// Mitsubishi GX Works2 project: DALG_TRAM_BE_TONG_ANALOG   PLC: FX3U/FX3UC

PROGRAM MAIN
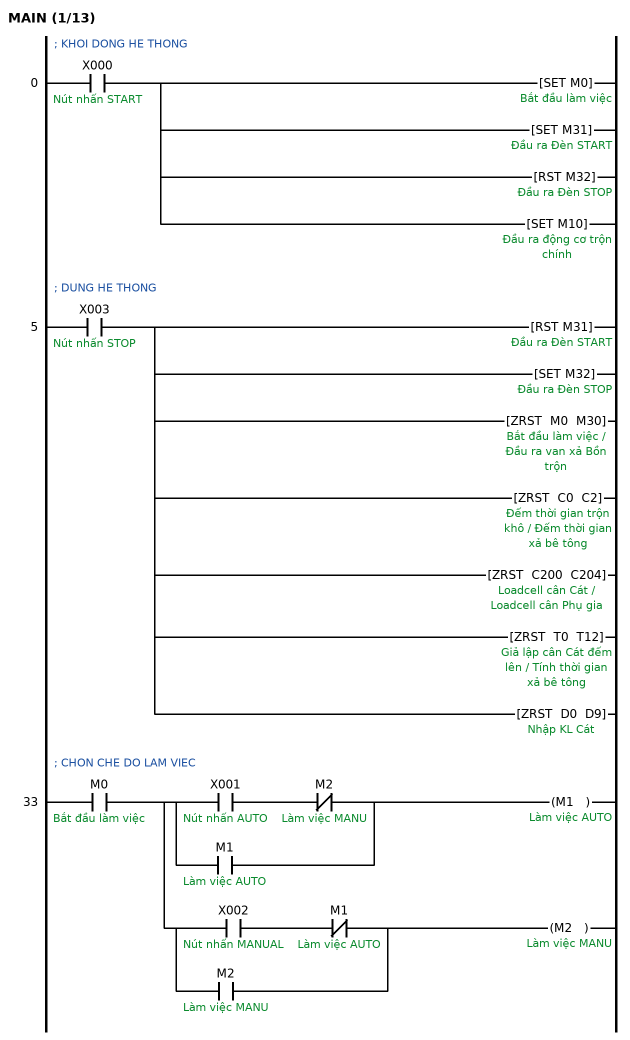
; KHOI DONG HE THONG
0     LD      X000  ; Nút nhấn START
      SET     M0  ; Bắt đầu làm việc
      SET     M31  ; Đầu ra Đèn START
      RST     M32  ; Đầu ra Đèn STOP
      SET     M10  ; Đầu ra động cơ trộn chính
; DUNG HE THONG
5     LD      X003  ; Nút nhấn STOP
      RST     M31  ; Đầu ra Đèn START
      SET     M32  ; Đầu ra Đèn STOP
      ZRST    M0 M30  ; Đầu ra van xả Bồn trộn
      ZRST    C0 C2  ; Đếm thời gian trộn khô / Đếm thời gian xả bê tông
      ZRST    C200 C204  ; Loadcell cân Cát / Loadcell cân Phụ gia
      ZRST    T0 T12  ; Giả lập cân Cát đếm lên / Tính thời gian xả bê tông
      ZRST    D0 D9  ; Nhập KL Cát
; CHON CHE DO LAM VIEC
33    LD      M0  ; Bắt đầu làm việc
      MPS
      LD      X001  ; Nút nhấn AUTO
      ANI     M2  ; Làm việc MANU
      OR      M1  ; Làm việc AUTO
      ANB
      OUT     M1  ; Làm việc AUTO
      MPP
      LD      X002  ; Nút nhấn MANUAL
      ANI     M1  ; Làm việc AUTO
      OR      M2  ; Làm việc MANU
      ANB
      OUT     M2  ; Làm việc MANU
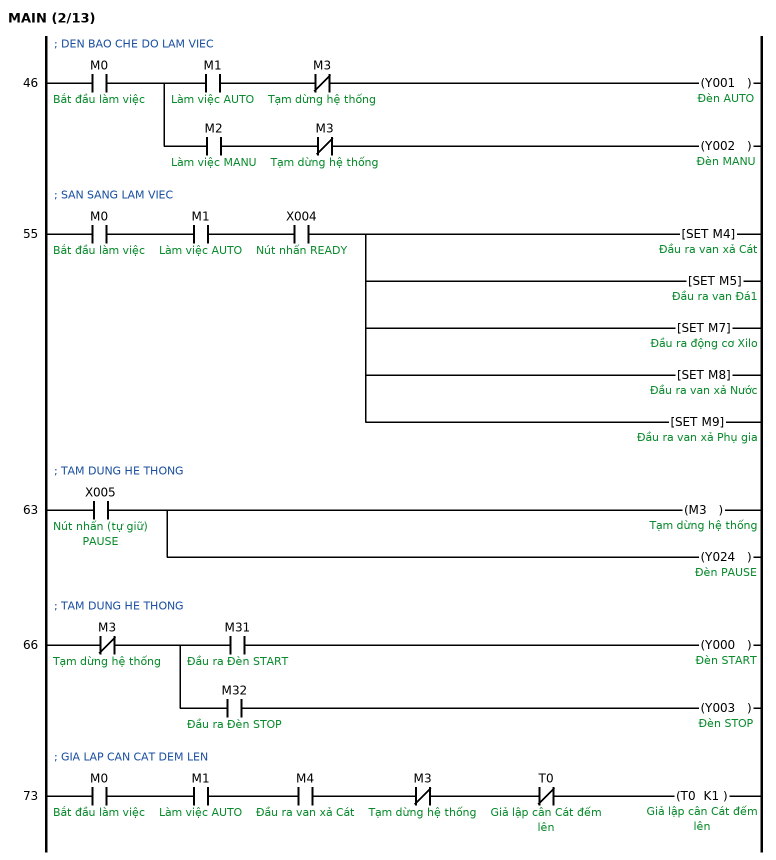
; DEN BAO CHE DO LAM VIEC
46    LD      M0  ; Bắt đầu làm việc
      MPS
      AND     M1  ; Làm việc AUTO
      ANI     M3  ; Tạm dừng hệ thống
      OUT     Y001  ; Đèn AUTO
      MPP
      AND     M2  ; Làm việc MANU
      ANI     M3  ; Tạm dừng hệ thống
      OUT     Y002  ; Đèn MANU
; SAN SANG LAM VIEC
55    LD      M0  ; Bắt đầu làm việc
      AND     M1  ; Làm việc AUTO
      AND     X004  ; Nút nhấn READY
      SET     M4  ; Đầu ra van xả Cát
      SET     M5  ; Đầu ra van Đá1
      SET     M7  ; Đầu ra động cơ Xilo
      SET     M8  ; Đầu ra van xả Nước
      SET     M9  ; Đầu ra van xả Phụ gia
; TAM DUNG HE THONG
63    LD      X005  ; Nút nhấn (tự giữ) PAUSE
      OUT     M3  ; Tạm dừng hệ thống
      OUT     Y024  ; Đèn PAUSE
; TAM DUNG HE THONG
66    LDI     M3  ; Tạm dừng hệ thống
      MPS
      AND     M31  ; Đầu ra Đèn START
      OUT     Y000  ; Đèn START
      MPP
      AND     M32  ; Đầu ra Đèn STOP
      OUT     Y003  ; Đèn STOP
; GIA LAP CAN CAT DEM LEN
73    LD      M0  ; Bắt đầu làm việc
      AND     M1  ; Làm việc AUTO
      AND     M4  ; Đầu ra van xả Cát
      ANI     M3  ; Tạm dừng hệ thống
      ANI     T0  ; Giả lập cân Cát đếm lên
      OUT     T0 K1  ; Giả lập cân Cát đếm lên
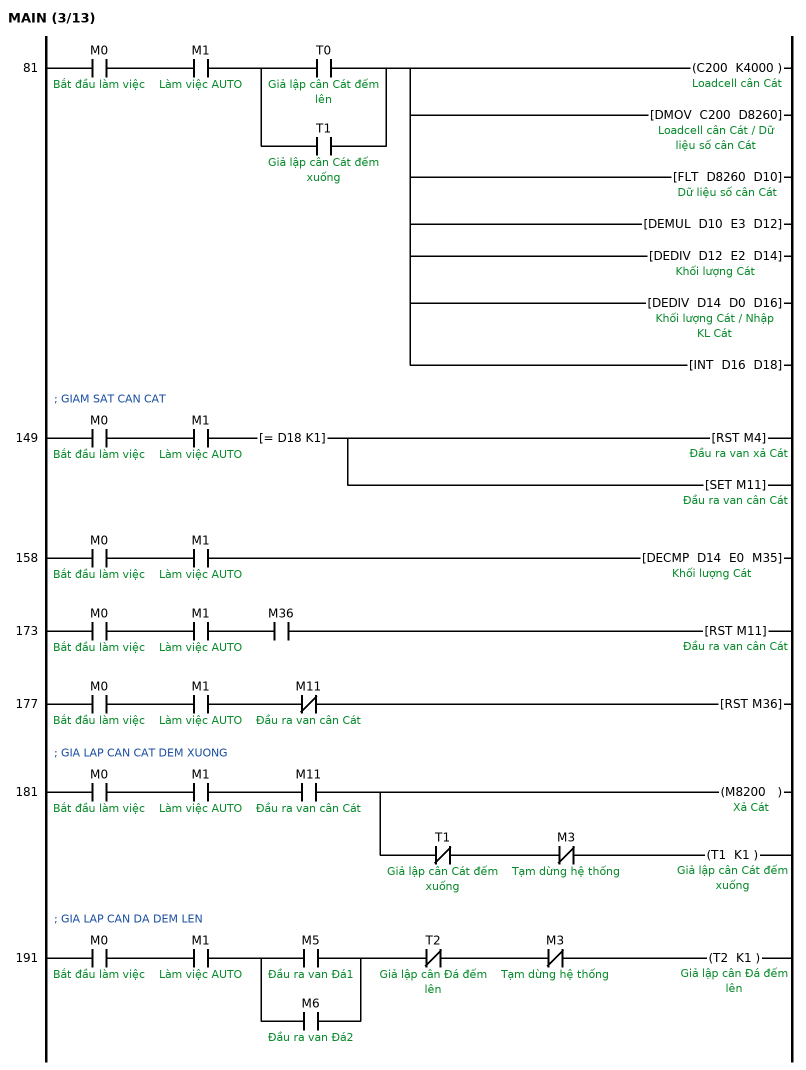
81    LD      M0  ; Bắt đầu làm việc
      AND     M1  ; Làm việc AUTO
      LD      T0  ; Giả lập cân Cát đếm lên
      OR      T1  ; Giả lập cân Cát đếm xuống
      ANB
      OUT     C200 K4000  ; Loadcell cân Cát
      DMOV    C200 D8260  ; Dữ liệu số cân Cát
      FLT     D8260 D10
      DEMUL   D10 E3 D12
      DEDIV   D12 E2 D14  ; Khối lượng Cát
      DEDIV   D14 D0 D16
      INT     D16 D18
; GIAM SAT CAN CAT
149   LD      M0  ; Bắt đầu làm việc
      AND     M1  ; Làm việc AUTO
      AND=    D18 K1
      RST     M4  ; Đầu ra van xả Cát
      SET     M11  ; Đầu ra van cân Cát
158   LD      M0  ; Bắt đầu làm việc
      AND     M1  ; Làm việc AUTO
      DECMP   D14 E0 M35
173   LD      M0  ; Bắt đầu làm việc
      AND     M1  ; Làm việc AUTO
      AND     M36
      RST     M11  ; Đầu ra van cân Cát
177   LD      M0  ; Bắt đầu làm việc
      AND     M1  ; Làm việc AUTO
      ANI     M11  ; Đầu ra van cân Cát
      RST     M36
; GIA LAP CAN CAT DEM XUONG
181   LD      M0  ; Bắt đầu làm việc
      AND     M1  ; Làm việc AUTO
      AND     M11  ; Đầu ra van cân Cát
      OUT     M8200  ; Xả Cát
      ANI     T1  ; Giả lập cân Cát đếm xuống
      ANI     M3  ; Tạm dừng hệ thống
      OUT     T1 K1  ; Giả lập cân Cát đếm xuống
; GIA LAP CAN DA DEM LEN
191   LD      M0  ; Bắt đầu làm việc
      AND     M1  ; Làm việc AUTO
      LD      M5  ; Đầu ra van Đá1
      OR      M6  ; Đầu ra van Đá2
      ANB
      ANI     T2  ; Giả lập cân Đá đếm lên
      ANI     M3  ; Tạm dừng hệ thống
      OUT     T2 K1  ; Giả lập cân Đá đếm lên
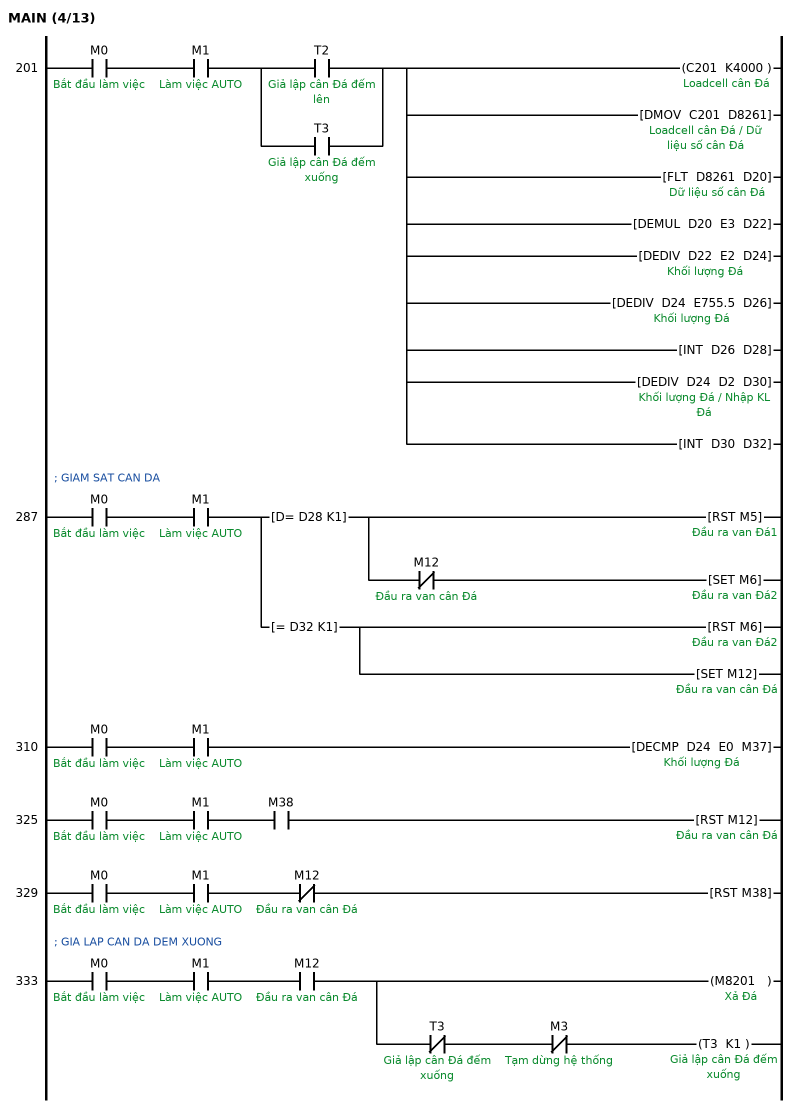
201   LD      M0  ; Bắt đầu làm việc
      AND     M1  ; Làm việc AUTO
      LD      T2  ; Giả lập cân Đá đếm lên
      OR      T3  ; Giả lập cân Đá đếm xuống
      ANB
      OUT     C201 K4000  ; Loadcell cân Đá
      DMOV    C201 D8261  ; Dữ liệu số cân Đá
      FLT     D8261 D20
      DEMUL   D20 E3 D22
      DEDIV   D22 E2 D24  ; Khối lượng Đá
      DEDIV   D24 E755.5 D26
      INT     D26 D28
      DEDIV   D24 D2 D30  ; Nhập KL Đá
      INT     D30 D32
; GIAM SAT CAN DA
287   LD      M0  ; Bắt đầu làm việc
      AND     M1  ; Làm việc AUTO
      MPS
      ANDD=   D28 K1
      RST     M5  ; Đầu ra van Đá1
      ANI     M12  ; Đầu ra van cân Đá
      SET     M6  ; Đầu ra van Đá2
      MPP
      AND=    D32 K1
      RST     M6  ; Đầu ra van Đá2
      SET     M12  ; Đầu ra van cân Đá
310   LD      M0  ; Bắt đầu làm việc
      AND     M1  ; Làm việc AUTO
      DECMP   D24 E0 M37
325   LD      M0  ; Bắt đầu làm việc
      AND     M1  ; Làm việc AUTO
      AND     M38
      RST     M12  ; Đầu ra van cân Đá
329   LD      M0  ; Bắt đầu làm việc
      AND     M1  ; Làm việc AUTO
      ANI     M12  ; Đầu ra van cân Đá
      RST     M38
; GIA LAP CAN DA DEM XUONG
333   LD      M0  ; Bắt đầu làm việc
      AND     M1  ; Làm việc AUTO
      AND     M12  ; Đầu ra van cân Đá
      OUT     M8201  ; Xả Đá
      ANI     T3  ; Giả lập cân Đá đếm xuống
      ANI     M3  ; Tạm dừng hệ thống
      OUT     T3 K1  ; Giả lập cân Đá đếm xuống
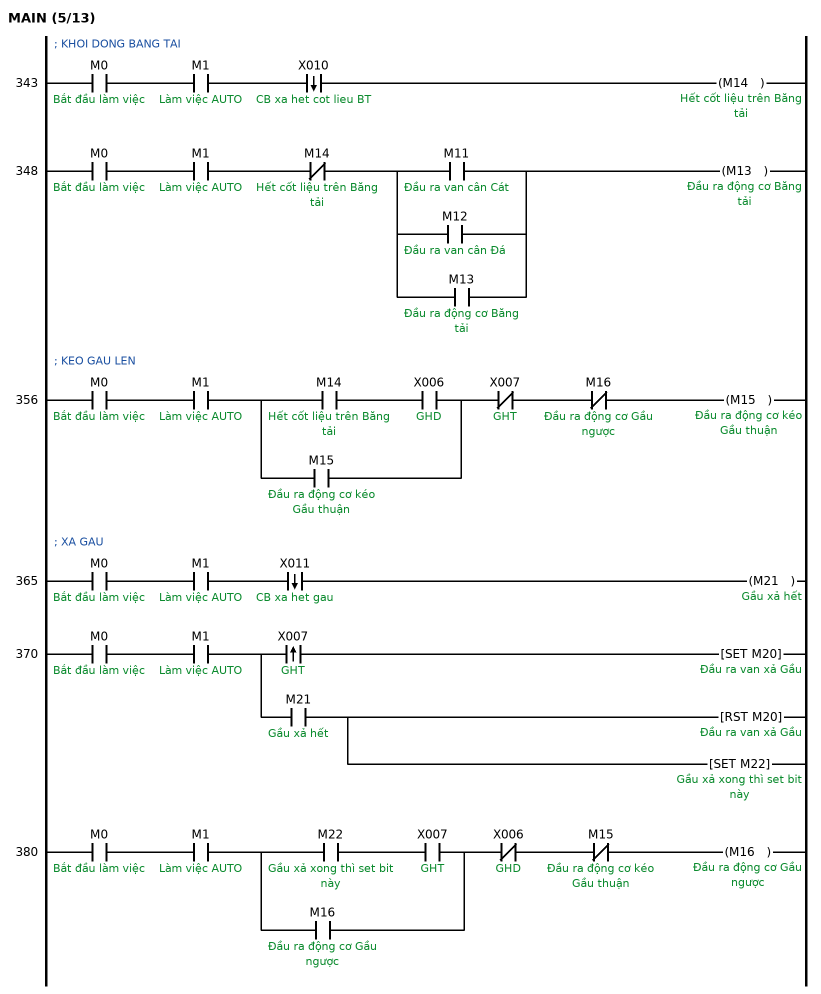
; KHOI DONG BANG TAI
343   LD      M0  ; Bắt đầu làm việc
      AND     M1  ; Làm việc AUTO
      ANDF    X010  ; CB xa het cot lieu BT
      OUT     M14  ; Hết cốt liệu trên Băng tải
348   LD      M0  ; Bắt đầu làm việc
      AND     M1  ; Làm việc AUTO
      ANI     M14  ; Hết cốt liệu trên Băng tải
      LD      M11  ; Đầu ra van cân Cát
      OR      M12  ; Đầu ra van cân Đá
      OR      M13  ; Đầu ra động cơ Băng tải
      ANB
      OUT     M13  ; Đầu ra động cơ Băng tải
; KEO GAU LEN
356   LD      M0  ; Bắt đầu làm việc
      AND     M1  ; Làm việc AUTO
      LD      M14  ; Hết cốt liệu trên Băng tải
      AND     X006  ; GHD
      OR      M15  ; Đầu ra động cơ kéo Gầu thuận
      ANB
      ANI     X007  ; GHT
      ANI     M16  ; Đầu ra động cơ Gầu ngược
      OUT     M15  ; Đầu ra động cơ kéo Gầu thuận
; XA GAU
365   LD      M0  ; Bắt đầu làm việc
      AND     M1  ; Làm việc AUTO
      ANDF    X011  ; CB xa het gau
      OUT     M21  ; Gầu xả hết
370   LD      M0  ; Bắt đầu làm việc
      AND     M1  ; Làm việc AUTO
      MPS
      ANDP    X007  ; GHT
      SET     M20  ; Đầu ra van xả Gầu
      MPP
      AND     M21  ; Gầu xả hết
      RST     M20  ; Đầu ra van xả Gầu
      SET     M22  ; Gầu xả xong thì set bit này
380   LD      M0  ; Bắt đầu làm việc
      AND     M1  ; Làm việc AUTO
      LD      M22  ; Gầu xả xong thì set bit này
      AND     X007  ; GHT
      OR      M16  ; Đầu ra động cơ Gầu ngược
      ANB
      ANI     X006  ; GHD
      ANI     M15  ; Đầu ra động cơ kéo Gầu thuận
      OUT     M16  ; Đầu ra động cơ Gầu ngược
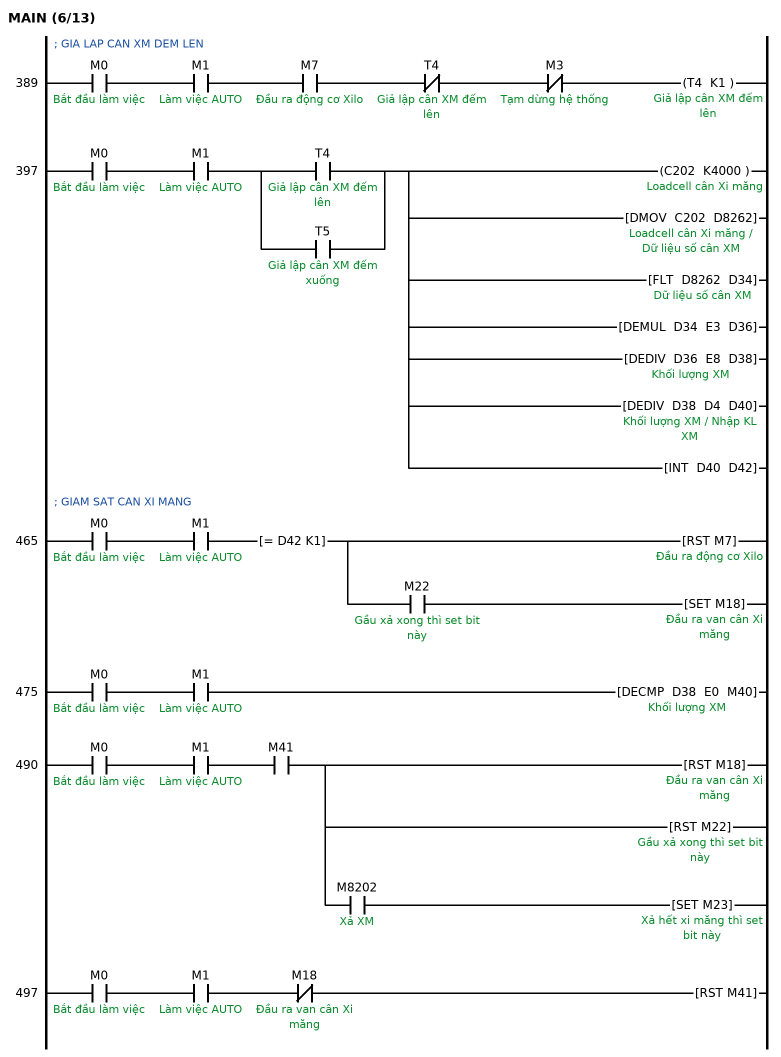
; GIA LAP CAN XM DEM LEN
389   LD      M0  ; Bắt đầu làm việc
      AND     M1  ; Làm việc AUTO
      AND     M7  ; Đầu ra động cơ Xilo
      ANI     T4  ; Giả lập cân XM đếm lên
      ANI     M3  ; Tạm dừng hệ thống
      OUT     T4 K1  ; Giả lập cân XM đếm lên
397   LD      M0  ; Bắt đầu làm việc
      AND     M1  ; Làm việc AUTO
      LD      T4  ; Giả lập cân XM đếm lên
      OR      T5  ; Giả lập cân XM đếm xuống
      ANB
      OUT     C202 K4000  ; Loadcell cân Xi măng
      DMOV    C202 D8262  ; Dữ liệu số cân XM
      FLT     D8262 D34
      DEMUL   D34 E3 D36
      DEDIV   D36 E8 D38  ; Khối lượng XM
      DEDIV   D38 D4 D40  ; Nhập KL XM
      INT     D40 D42
; GIAM SAT CAN XI MANG
465   LD      M0  ; Bắt đầu làm việc
      AND     M1  ; Làm việc AUTO
      AND=    D42 K1
      RST     M7  ; Đầu ra động cơ Xilo
      AND     M22  ; Gầu xả xong thì set bit này
      SET     M18  ; Đầu ra van cân Xi măng
475   LD      M0  ; Bắt đầu làm việc
      AND     M1  ; Làm việc AUTO
      DECMP   D38 E0 M40
490   LD      M0  ; Bắt đầu làm việc
      AND     M1  ; Làm việc AUTO
      AND     M41
      RST     M18  ; Đầu ra van cân Xi măng
      RST     M22  ; Gầu xả xong thì set bit này
      AND     M8202  ; Xả XM
      SET     M23  ; Xả hết xi măng thì set bit này
497   LD      M0  ; Bắt đầu làm việc
      AND     M1  ; Làm việc AUTO
      ANI     M18  ; Đầu ra van cân Xi măng
      RST     M41
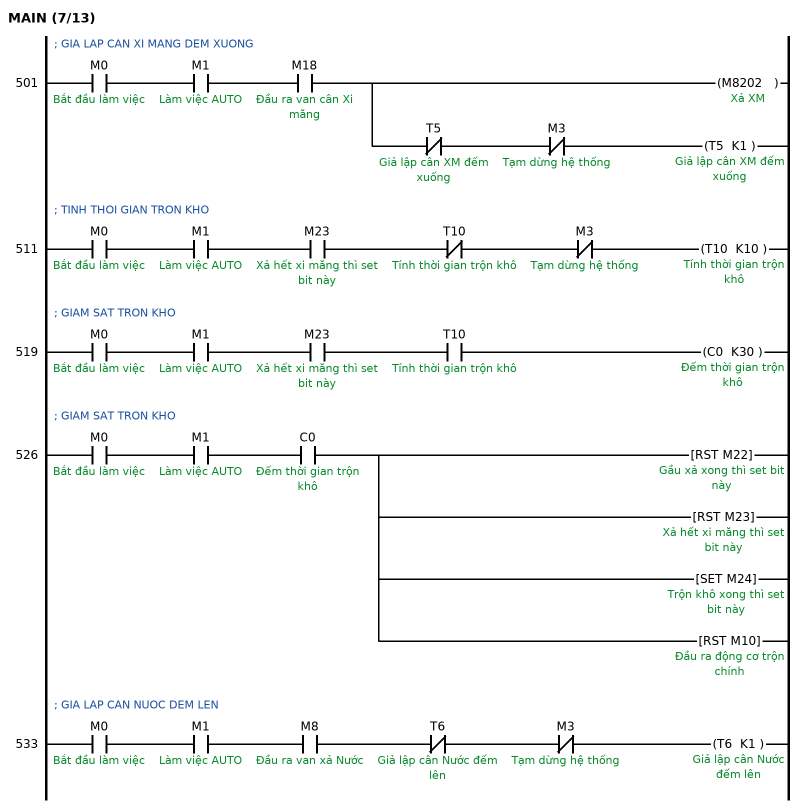
; GIA LAP CAN XI MANG DEM XUONG
501   LD      M0  ; Bắt đầu làm việc
      AND     M1  ; Làm việc AUTO
      AND     M18  ; Đầu ra van cân Xi măng
      OUT     M8202  ; Xả XM
      ANI     T5  ; Giả lập cân XM đếm xuống
      ANI     M3  ; Tạm dừng hệ thống
      OUT     T5 K1  ; Giả lập cân XM đếm xuống
; TINH THOI GIAN TRON KHO
511   LD      M0  ; Bắt đầu làm việc
      AND     M1  ; Làm việc AUTO
      AND     M23  ; Xả hết xi măng thì set bit này
      ANI     T10  ; Tính thời gian trộn khô
      ANI     M3  ; Tạm dừng hệ thống
      OUT     T10 K10  ; Tính thời gian trộn khô
; GIAM SAT TRON KHO
519   LD      M0  ; Bắt đầu làm việc
      AND     M1  ; Làm việc AUTO
      AND     M23  ; Xả hết xi măng thì set bit này
      AND     T10  ; Tính thời gian trộn khô
      OUT     C0 K30  ; Đếm thời gian trộn khô
; GIAM SAT TRON KHO
526   LD      M0  ; Bắt đầu làm việc
      AND     M1  ; Làm việc AUTO
      AND     C0  ; Đếm thời gian trộn khô
      RST     M22  ; Gầu xả xong thì set bit này
      RST     M23  ; Xả hết xi măng thì set bit này
      SET     M24  ; Trộn khô xong thì set bit này
      RST     M10  ; Đầu ra động cơ trộn chính
; GIA LAP CAN NUOC DEM LEN
533   LD      M0  ; Bắt đầu làm việc
      AND     M1  ; Làm việc AUTO
      AND     M8  ; Đầu ra van xả Nước
      ANI     T6  ; Giả lập cân Nước đếm lên
      ANI     M3  ; Tạm dừng hệ thống
      OUT     T6 K1  ; Giả lập cân Nước đếm lên
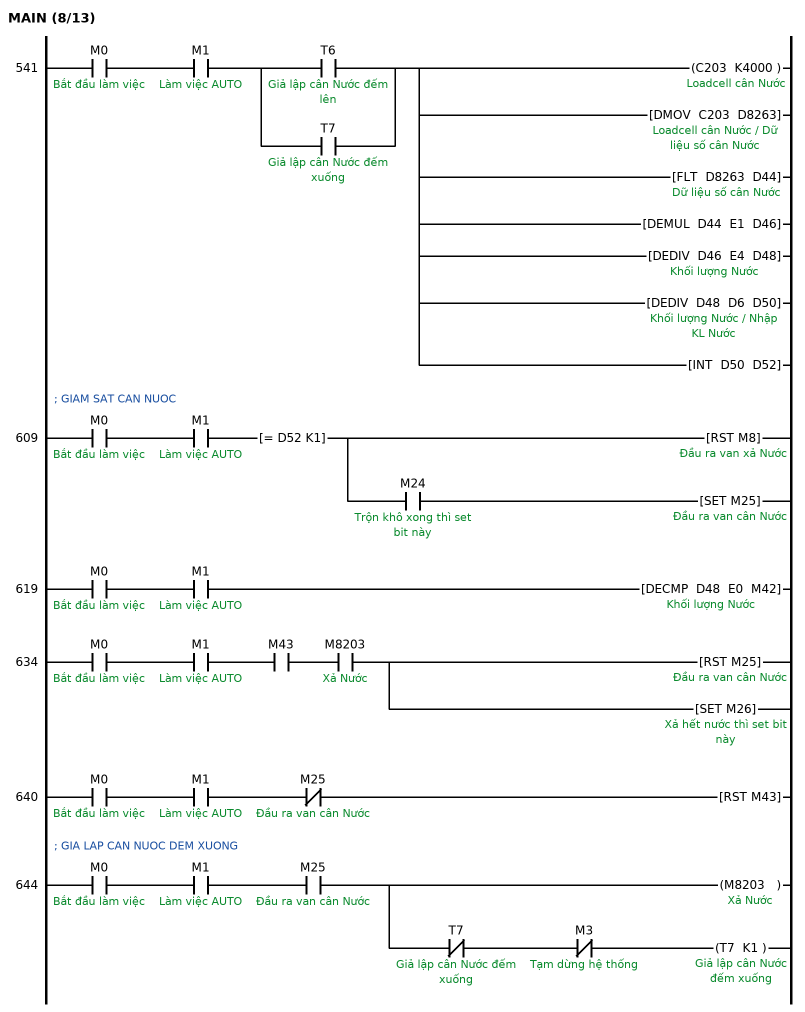
541   LD      M0  ; Bắt đầu làm việc
      AND     M1  ; Làm việc AUTO
      LD      T6  ; Giả lập cân Nước đếm lên
      OR      T7  ; Giả lập cân Nước đếm xuống
      ANB
      OUT     C203 K4000  ; Loadcell cân Nước
      DMOV    C203 D8263  ; Dữ liệu số cân Nước
      FLT     D8263 D44
      DEMUL   D44 E1 D46
      DEDIV   D46 E4 D48  ; Khối lượng Nước
      DEDIV   D48 D6 D50  ; Nhập KL Nước
      INT     D50 D52
; GIAM SAT CAN NUOC
609   LD      M0  ; Bắt đầu làm việc
      AND     M1  ; Làm việc AUTO
      AND=    D52 K1
      RST     M8  ; Đầu ra van xả Nước
      AND     M24  ; Trộn khô xong thì set bit này
      SET     M25  ; Đầu ra van cân Nước
619   LD      M0  ; Bắt đầu làm việc
      AND     M1  ; Làm việc AUTO
      DECMP   D48 E0 M42
634   LD      M0  ; Bắt đầu làm việc
      AND     M1  ; Làm việc AUTO
      AND     M43
      AND     M8203  ; Xả Nước
      RST     M25  ; Đầu ra van cân Nước
      SET     M26  ; Xả hết nước thì set bit này
640   LD      M0  ; Bắt đầu làm việc
      AND     M1  ; Làm việc AUTO
      ANI     M25  ; Đầu ra van cân Nước
      RST     M43
; GIA LAP CAN NUOC DEM XUONG
644   LD      M0  ; Bắt đầu làm việc
      AND     M1  ; Làm việc AUTO
      AND     M25  ; Đầu ra van cân Nước
      OUT     M8203  ; Xả Nước
      ANI     T7  ; Giả lập cân Nước đếm xuống
      ANI     M3  ; Tạm dừng hệ thống
      OUT     T7 K1  ; Giả lập cân Nước đếm xuống
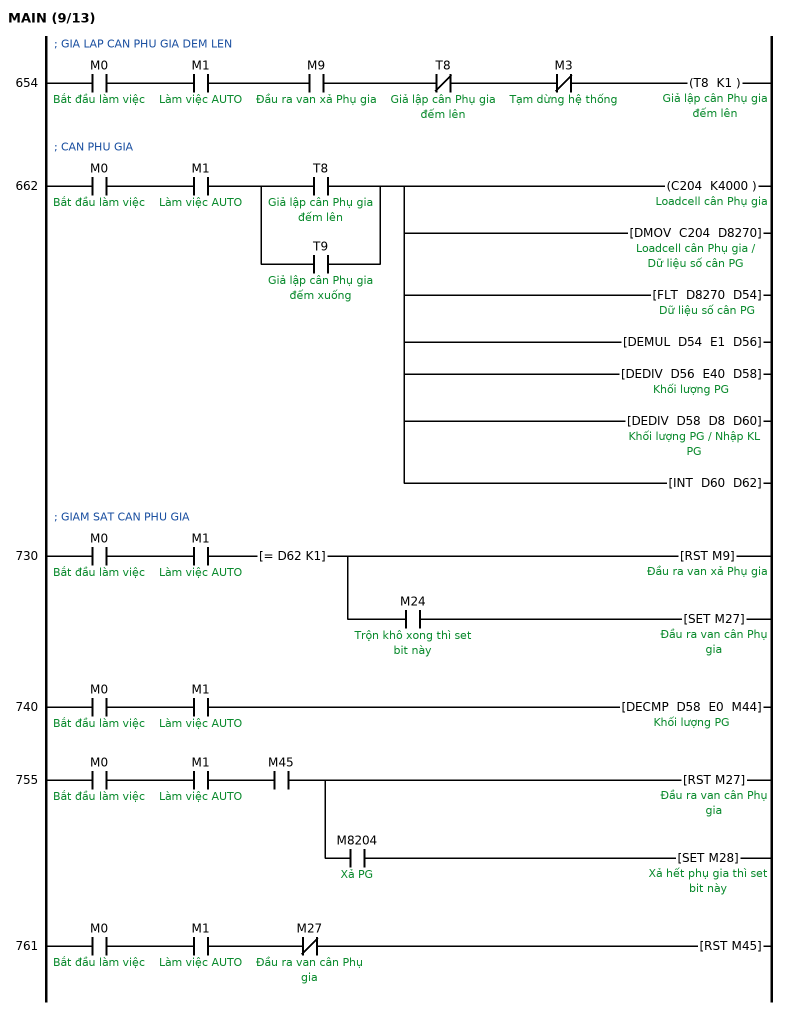
; GIA LAP CAN PHU GIA DEM LEN
654   LD      M0  ; Bắt đầu làm việc
      AND     M1  ; Làm việc AUTO
      AND     M9  ; Đầu ra van xả Phụ gia
      ANI     T8  ; Giả lập cân Phụ gia đếm lên
      ANI     M3  ; Tạm dừng hệ thống
      OUT     T8 K1  ; Giả lập cân Phụ gia đếm lên
; CAN PHU GIA
662   LD      M0  ; Bắt đầu làm việc
      AND     M1  ; Làm việc AUTO
      LD      T8  ; Giả lập cân Phụ gia đếm lên
      OR      T9  ; Giả lập cân Phụ gia đếm xuống
      ANB
      OUT     C204 K4000  ; Loadcell cân Phụ gia
      DMOV    C204 D8270  ; Dữ liệu số cân PG
      FLT     D8270 D54
      DEMUL   D54 E1 D56
      DEDIV   D56 E40 D58  ; Khối lượng PG
      DEDIV   D58 D8 D60  ; Nhập KL PG
      INT     D60 D62
; GIAM SAT CAN PHU GIA
730   LD      M0  ; Bắt đầu làm việc
      AND     M1  ; Làm việc AUTO
      AND=    D62 K1
      RST     M9  ; Đầu ra van xả Phụ gia
      AND     M24  ; Trộn khô xong thì set bit này
      SET     M27  ; Đầu ra van cân Phụ gia
740   LD      M0  ; Bắt đầu làm việc
      AND     M1  ; Làm việc AUTO
      DECMP   D58 E0 M44
755   LD      M0  ; Bắt đầu làm việc
      AND     M1  ; Làm việc AUTO
      AND     M45
      RST     M27  ; Đầu ra van cân Phụ gia
      AND     M8204  ; Xả PG
      SET     M28  ; Xả hết phụ gia thì set bit này
761   LD      M0  ; Bắt đầu làm việc
      AND     M1  ; Làm việc AUTO
      ANI     M27  ; Đầu ra van cân Phụ gia
      RST     M45
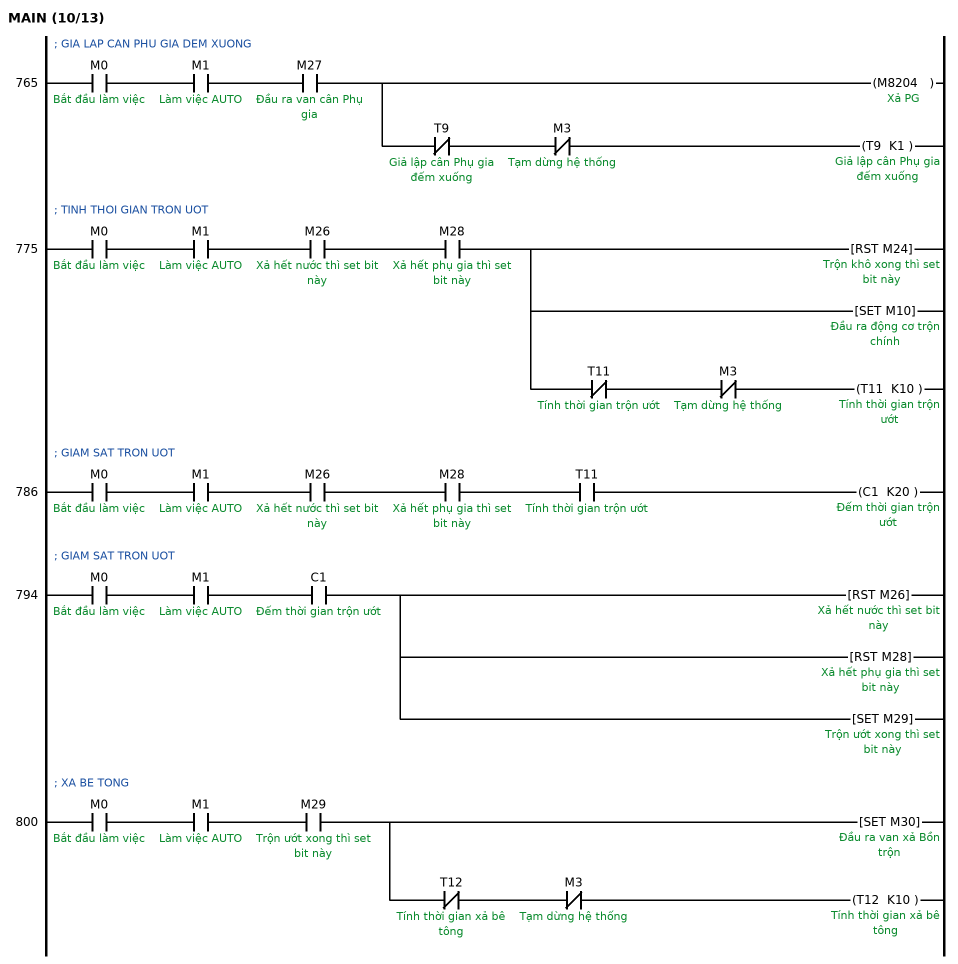
; GIA LAP CAN PHU GIA DEM XUONG
765   LD      M0  ; Bắt đầu làm việc
      AND     M1  ; Làm việc AUTO
      AND     M27  ; Đầu ra van cân Phụ gia
      OUT     M8204  ; Xả PG
      ANI     T9  ; Giả lập cân Phụ gia đếm xuống
      ANI     M3  ; Tạm dừng hệ thống
      OUT     T9 K1  ; Giả lập cân Phụ gia đếm xuống
; TINH THOI GIAN TRON UOT
775   LD      M0  ; Bắt đầu làm việc
      AND     M1  ; Làm việc AUTO
      AND     M26  ; Xả hết nước thì set bit này
      AND     M28  ; Xả hết phụ gia thì set bit này
      RST     M24  ; Trộn khô xong thì set bit này
      SET     M10  ; Đầu ra động cơ trộn chính
      ANI     T11  ; Tính thời gian trộn ướt
      ANI     M3  ; Tạm dừng hệ thống
      OUT     T11 K10  ; Tính thời gian trộn ướt
; GIAM SAT TRON UOT
786   LD      M0  ; Bắt đầu làm việc
      AND     M1  ; Làm việc AUTO
      AND     M26  ; Xả hết nước thì set bit này
      AND     M28  ; Xả hết phụ gia thì set bit này
      AND     T11  ; Tính thời gian trộn ướt
      OUT     C1 K20  ; Đếm thời gian trộn ướt
; GIAM SAT TRON UOT
794   LD      M0  ; Bắt đầu làm việc
      AND     M1  ; Làm việc AUTO
      AND     C1  ; Đếm thời gian trộn ướt
      RST     M26  ; Xả hết nước thì set bit này
      RST     M28  ; Xả hết phụ gia thì set bit này
      SET     M29  ; Trộn ướt xong thì set bit này
; XA BE TONG
800   LD      M0  ; Bắt đầu làm việc
      AND     M1  ; Làm việc AUTO
      AND     M29  ; Trộn ướt xong thì set bit này
      SET     M30  ; Đầu ra van xả Bồn trộn
      ANI     T12  ; Tính thời gian xả bê tông
      ANI     M3  ; Tạm dừng hệ thống
      OUT     T12 K10  ; Tính thời gian xả bê tông
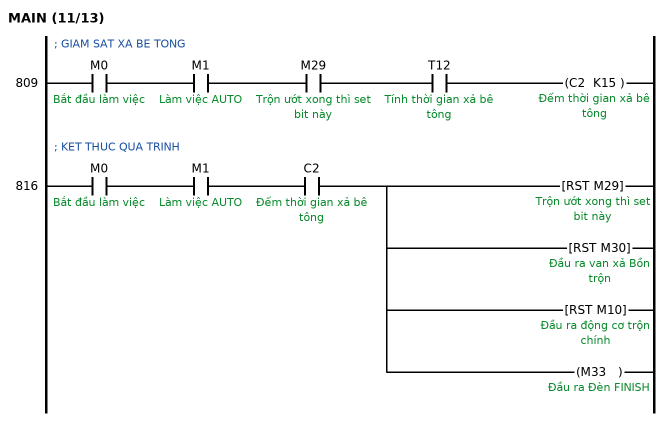
; GIAM SAT XA BE TONG
809   LD      M0  ; Bắt đầu làm việc
      AND     M1  ; Làm việc AUTO
      AND     M29  ; Trộn ướt xong thì set bit này
      AND     T12  ; Tính thời gian xả bê tông
      OUT     C2 K15  ; Đếm thời gian xả bê tông
; KET THUC QUA TRINH
816   LD      M0  ; Bắt đầu làm việc
      AND     M1  ; Làm việc AUTO
      AND     C2  ; Đếm thời gian xả bê tông
      RST     M29  ; Trộn ướt xong thì set bit này
      RST     M30  ; Đầu ra van xả Bồn trộn
      RST     M10  ; Đầu ra động cơ trộn chính
      OUT     M33  ; Đầu ra Đèn FINISH
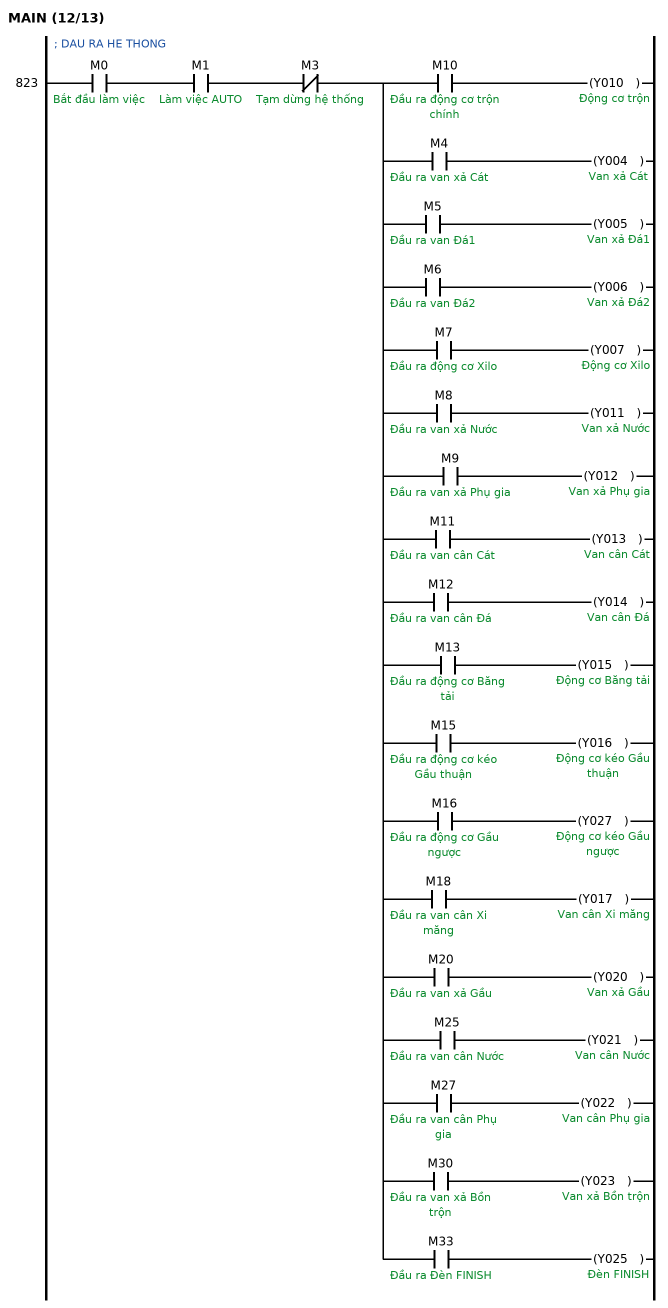
; DAU RA HE THONG
823   LD      M0  ; Bắt đầu làm việc
      AND     M1  ; Làm việc AUTO
      ANI     M3  ; Tạm dừng hệ thống
      MPS
      AND     M10  ; Đầu ra động cơ trộn chính
      OUT     Y010  ; Động cơ trộn
      MRD
      AND     M4  ; Đầu ra van xả Cát
      OUT     Y004  ; Van xả Cát
      MRD
      AND     M5  ; Đầu ra van Đá1
      OUT     Y005  ; Van xả Đá1
      MRD
      AND     M6  ; Đầu ra van Đá2
      OUT     Y006  ; Van xả Đá2
      MRD
      AND     M7  ; Đầu ra động cơ Xilo
      OUT     Y007  ; Động cơ Xilo
      MRD
      AND     M8  ; Đầu ra van xả Nước
      OUT     Y011  ; Van xả Nước
      MRD
      AND     M9  ; Đầu ra van xả Phụ gia
      OUT     Y012  ; Van xả Phụ gia
      MRD
      AND     M11  ; Đầu ra van cân Cát
      OUT     Y013  ; Van cân Cát
      MRD
      AND     M12  ; Đầu ra van cân Đá
      OUT     Y014  ; Van cân Đá
      MRD
      AND     M13  ; Đầu ra động cơ Băng tải
      OUT     Y015  ; Động cơ Băng tải
      MRD
      AND     M15  ; Đầu ra động cơ kéo Gầu thuận
      OUT     Y016  ; Động cơ kéo Gầu thuận
      MRD
      AND     M16  ; Đầu ra động cơ Gầu ngược
      OUT     Y027  ; Động cơ kéo Gầu ngược
      MRD
      AND     M18  ; Đầu ra van cân Xi măng
      OUT     Y017  ; Van cân Xi măng
      MRD
      AND     M20  ; Đầu ra van xả Gầu
      OUT     Y020  ; Van xả Gầu
      MRD
      AND     M25  ; Đầu ra van cân Nước
      OUT     Y021  ; Van cân Nước
      MRD
      AND     M27  ; Đầu ra van cân Phụ gia
      OUT     Y022  ; Van cân Phụ gia
      MRD
      AND     M30  ; Đầu ra van xả Bồn trộn
      OUT     Y023  ; Van xả Bồn trộn
      MPP
      AND     M33  ; Đầu ra Đèn FINISH
      OUT     Y025  ; Đèn FINISH
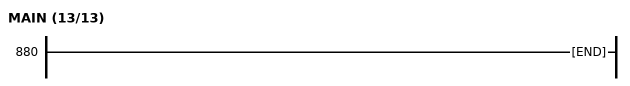
880   END
END_PROGRAM
